(* CoDeSys 2.3.9.62 project: Tema1 Ejemplo5-Cilindro2 v0.pro *)

(* Global variable list: Global_Variables *)
VAR_GLOBAL
  A:BOOL;
  B:BOOL;
  K1:BOOL;
  K2:BOOL;
 S1:BOOL;
END_VAR

(* POU PLC_PRG, ST *)
PROGRAM PLC_PRG
VAR
  posy:INT;
END_VAR
Control();


IF K1=TRUE THEN
IF posy<100 THEN
  posy:=posy+1;
END_IF
END_IF

IF K2=TRUE THEN
IF posy>0 THEN
  posy:=posy-1;
END_IF
END_IF


IF posy<=0 THEN
  A:=TRUE;
ELSE
  A:=FALSE;
END_IF

IF posy>=100 THEN
  B:=TRUE;
ELSE
  B:=FALSE;
END_IF
END_PROGRAM

(* POU Control, LD *)
PROGRAM Control
VAR
END_VAR
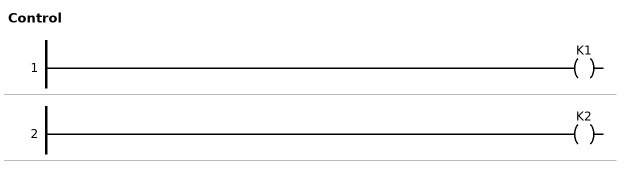
_LD_ (* Ladder Diagram *)
NETWORK 1
	* --- (K1)
NETWORK 2
	* --- (K2)
_END_LD_
(* the same logic as Structured Text *)
(* Network 1 *)
K1 := TRUE;
(* Network 2 *)
K2 := TRUE;
END_PROGRAM

(* Visualisation Deposito
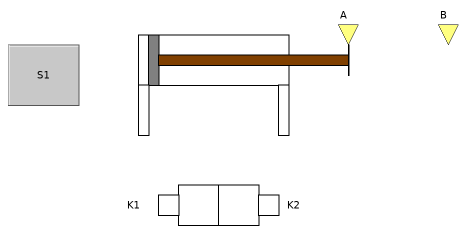
button at (50,80)-(121,141): text "S1"; taps .S1
polygon at (380,60)-(400,80): alarm colour if .A; toggles .B
rectangle at (190,70)-(201,121): left PLC_PRG.posy; right PLC_PRG.posy
rectangle at (200,90)-(391,101): left PLC_PRG.posy; right PLC_PRG.posy
polygon at (480,60)-(500,80): alarm colour if .B; toggles .B
rectangle at (390,80)-(391,111): left PLC_PRG.posy; right PLC_PRG.posy
rectangle at (220,220)-(261,261): alarm colour if .K1
rectangle at (260,220)-(301,261): alarm colour if .K2
rectangle at (200,230)-(221,251): alarm colour if .K1
rectangle at (180,120)-(191,171): alarm colour if .K1
rectangle at (320,120)-(331,171): alarm colour if .K2
rectangle at (300,230)-(321,251): alarm colour if .K2
rectangle at (310,220)-(361,261): text "K2"
rectangle at (150,220)-(201,261): text "K1"
rectangle at (360,30)-(411,71): text "A"
rectangle at (460,30)-(511,71): text "B"
1 more shapes without text or variables
*)
